// SIMATIC S7-200 project (STEP 7-Micro/WIN), CPU 226 REL 02.01

SYMBOL_TABLE SYM1
ADDR_H           VB102
ADDR_L           VB103
D_H              VB114
D_L              VB115
DATA2_H          VB118
DATA2_L          VB119
DATA1_H          VB120
DATA1_L          VB121
SUM_H            VB122
SUM_L            VB123
SADDR_H          VW202
SADDR_L          VW204
S46H             VW206
S46L             VW208
S51              VW210
S57              VW212
S30_1            VW214
S44              VW216
S30_2            VW218
S30_3            VW220
S30_4            VW222
S30_5            VW224
SD_L             VW226
SD_H             VW228
S30_6            VW230
S31              VW232
SDATA2_H         VW234
SDATA2_L         VW236
SDATA1_H         VW238
SDATA1_L         VW240
END_SYMBOL_TABLE

ORGANIZATION_BLOCK OB_1:OB1
TITLE=【S7-200 PLC与DDM4A数显表的通信控制系统（二）】
// 在生产线上，PLC通过定时器以60个时间周期实现轮询控制。轮询时向分布在不同位置的16个DDM4A数显表发送计数数据，用于显示生产计数和设备状态等关键参数。
// 站点七作为生产线的核心区域，其的DDM4A数显表的计数数据根据实际检测量完成更新。此数据可供其他站点在需要时访问。
// 所有的DDM4A数显表配置为无校验、8位数据、波特率9600bps，使用自由口协议。发送缓冲区长度设为23字节。PLC串口设置和发送缓冲区与之保持一致，以确保通讯正常。
// 在主程序中，首先通过首次扫描设置串口控制字节，启用自由口模式，同时将发送缓冲区长度设为23字节，并初始化轮询控制变量为+1。
// 通过始终为1的位调用轮询子程序。轮询子程序中定时器每60个时间周期触发一次，触发时轮询控制变量左移一位，用于控制轮询。
// 主程序的多个网络分别对应1#站到16#站的发送逻辑。例如，当某站触发信号为真时，设置地址和数据字节，然后调用发送子程序。其他站的逻辑类似，只是地址字节依次递增，最后一站地址使用特定组合。在发送触发网络中，检测各站触发信号的上升沿，任何一位触发时，发送缓冲区开始的23字节数据。
// 在发送子程序中，设置发送缓冲区内容，例如多个命令字节作为固定命令代码。填充字节设为固定值，用于构成数据帧。后续网络将地址字节等转换为整数，存储在变量中，便于计算。校验网络计算SUM校验和，逐步累加所有相关字节的整数值。
// 校验处理网络中，将SUM低字节处理后转换为ASCII码，存储在临时位置，最终设置校验高低字节。
// 轮询子程序的控制网络中，当定时器触发时，轮询控制变量左移一位，实现轮询控制。定时网络中，如果定时器未触发，则启动定时器计时60个周期。
// 数据更新网络中，当站点七触发信号上升沿时，计数变量自增，若达到上限则重置为0，然后将计数变量转换为ASCII码，设置数据字节。
// 站触发信号逐一触发各站发送逻辑。通过触发信号的上升沿检测，确保同一时间只有一个站发送数据。串口配置为无校验、8位数据、波特率9600bps，使用自由口协议，与数显表保持一致。
BEGIN
Network 1
LD     SM0.1
MOVB   16#9, SMB30
MOVB   23, VB100
MOVW   +1, MW1
?000
Network 2
LD     SM0.0
CALL   SBR_1:SBR1
Network 3 // 发送1＃站数据
// 
// 
LD     M1.0
LPS
MOVB   16#31, ADDR_L:VB103
AENO
MOVB   16#30, ADDR_H:VB102
AENO
MOVB   16#30, D_L:VB115
AENO
MOVB   16#30, D_H:VB114
LPP
CALL   SBR_0:SBR0
Network 4 // 发送2＃站数据
// 
// 
LD     M1.1
LPS
MOVB   16#32, ADDR_L:VB103
AENO
MOVB   16#30, ADDR_H:VB102
LPP
CALL   SBR_0:SBR0
Network 5 // 发送3＃站数据
// 
// 
LD     M1.2
LPS
MOVB   16#33, ADDR_L:VB103
AENO
MOVB   16#30, ADDR_H:VB102
LPP
CALL   SBR_0:SBR0
Network 6 // 发送4＃站数据
// 
// 
LD     M1.3
LPS
MOVB   16#34, ADDR_L:VB103
AENO
MOVB   16#30, ADDR_H:VB102
LPP
CALL   SBR_0:SBR0
Network 7 // 发送5＃站数据
// 
// 
LD     M1.4
LPS
MOVB   16#35, ADDR_L:VB103
AENO
MOVB   16#30, ADDR_H:VB102
LPP
CALL   SBR_0:SBR0
Network 8 // 发送6＃站数据
// 
// 
LD     M1.5
LPS
MOVB   16#36, ADDR_L:VB103
AENO
MOVB   16#30, ADDR_H:VB102
LPP
CALL   SBR_0:SBR0
Network 9 // 发送7＃站数据
// 
// 
LD     M1.6
LPS
MOVB   16#37, ADDR_L:VB103
AENO
MOVB   16#30, ADDR_H:VB102
LPP
CALL   SBR_0:SBR0
Network 10 // 发送8＃站数据
// 
// 
LD     M1.7
LPS
MOVB   16#38, ADDR_L:VB103
AENO
MOVB   16#30, ADDR_H:VB102
LPP
CALL   SBR_0:SBR0
Network 11 // 发送9＃站数据
// 
// 
LD     M2.0
LPS
MOVB   16#39, ADDR_L:VB103
AENO
MOVB   16#30, ADDR_H:VB102
LPP
CALL   SBR_0:SBR0
Network 12 // 发送10＃站数据
// 
// 
LD     M2.1
LPS
MOVB   16#41, ADDR_L:VB103
AENO
MOVB   16#30, ADDR_H:VB102
LPP
CALL   SBR_0:SBR0
Network 13 // 发送11＃站数据
// 
// 
LD     M2.2
LPS
MOVB   16#42, ADDR_L:VB103
AENO
MOVB   16#30, ADDR_H:VB102
LPP
CALL   SBR_0:SBR0
Network 14 // 发送12＃站数据
// 
// 
LD     M2.3
LPS
MOVB   16#43, ADDR_L:VB103
AENO
MOVB   16#30, ADDR_H:VB102
LPP
CALL   SBR_0:SBR0
Network 15 // 发送13＃站数据
// 
// 
LD     M2.4
LPS
MOVB   16#44, ADDR_L:VB103
AENO
MOVB   16#30, ADDR_H:VB102
LPP
CALL   SBR_0:SBR0
Network 16 // 发送14＃站数据
// 
// 
LD     M2.5
LPS
MOVB   16#45, ADDR_L:VB103
AENO
MOVB   16#30, ADDR_H:VB102
LPP
CALL   SBR_0:SBR0
Network 17 // 发送15＃站数据
// 
// 
LD     M2.6
LPS
MOVB   16#46, ADDR_L:VB103
AENO
MOVB   16#30, ADDR_H:VB102
LPP
CALL   SBR_0:SBR0
Network 18 // 发送16＃站数据
// 
// 
LD     M2.7
LPS
MOVB   16#30, ADDR_L:VB103
AENO
MOVB   16#31, ADDR_H:VB102
LPP
CALL   SBR_0:SBR0
Network 19 // 发送程序
// 
// 
LD     M1.0
EU
LD     M1.1
EU
OLD
LD     M1.2
EU
OLD
LD     M1.3
EU
OLD
LD     M1.4
EU
OLD
LD     M1.5
EU
OLD
LD     M1.6
EU
OLD
LD     M1.7
EU
OLD
LD     M2.0
EU
OLD
LD     M2.1
EU
OLD
LD     M2.2
EU
OLD
LD     M2.3
EU
OLD
LD     M2.4
EU
OLD
LD     M2.5
EU
OLD
LD     M2.6
EU
OLD
LD     M2.7
EU
OLD
XMT    VB100, 0
END_ORGANIZATION_BLOCK

SUBROUTINE_BLOCK SBR_0:SBR0
TITLE=
BEGIN
Network 1 // 通讯缓冲区 VB102、VB103＝地址；VB114、VB115＝寄存器组；VB118～VB21＝数据；VB122、VB123＝SUM；
LD     SM0.0
MOVB   16#5, VB101
Network 2 // 计算机命令16#46H
//  
LD     SM0.0
MOVB   16#46, VB104
Network 3 // 计算机命令16#46L
//  
LD     SM0.0
MOVB   16#46, VB105
Network 4 // 16#51H
//  
LD     SM0.0
MOVB   16#51, VB106
Network 5 // 16#57
//  
LD     SM0.0
MOVB   16#57, VB107
Network 6 // 16#30
//  
LD     SM0.0
MOVB   16#30, VB108
Network 7 // 16#44
LD     SM0.0
MOVB   16#44, VB109
Network 8 // 16#30
//  
LD     SM0.0
MOVB   16#30, VB110
Network 9 // 16#30
LD     SM0.0
MOVB   16#30, VB111
Network 10 // 16#30
//  
LD     SM0.0
MOVB   16#30, VB112
Network 11 // 16#30
LD     SM0.0
MOVB   16#30, VB113
Network 12 // 16#30
//  
LD     SM0.0
MOVB   16#30, VB116
Network 13 // 16#31
//  
LD     SM0.0
MOVB   16#31, VB117
Network 14 // 将BYTE转换为整形数据，便于计算
LD     SM0.0
BTI    ADDR_L:VB103, SADDR_L:VW204
AENO
BTI    ADDR_H:VB102, SADDR_H:VW202
AENO
BTI    VB104, S46H:VW206
AENO
BTI    VB105, S46L:VW208
Network 15 // 将BYTE转换为整形数据，便于计算
LD     SM0.0
BTI    VB106, S51:VW210
AENO
BTI    VB107, S57:VW212
AENO
BTI    VB108, S30_1:VW214
AENO
BTI    VB109, S44:VW216
Network 16 // 将BYTE转换为整形数据，便于计算
LD     SM0.0
BTI    VB110, S30_2:VW218
AENO
BTI    VB111, S30_3:VW220
AENO
BTI    VB112, S30_4:VW222
AENO
BTI    VB113, S30_5:VW224
Network 17 // 将BYTE转换为整形数据，便于计算
LD     SM0.0
BTI    D_L:VB115, SD_L:VW226
AENO
BTI    D_H:VB114, SD_H:VW228
AENO
BTI    VB116, S30_6:VW230
AENO
BTI    VB117, S31:VW232
Network 18 // 将BYTE转换为整形数据，便于计算
// 
// 
LD     SM0.0
BTI    DATA2_L:VB119, SDATA2_L:VW236
AENO
BTI    DATA2_H:VB118, SDATA2_H:VW234
AENO
BTI    DATA1_L:VB121, SDATA1_L:VW240
AENO
BTI    DATA1_H:VB120, SDATA1_H:VW238
Network 19 // SUM计算
// 
// 
LD     SM0.0
MOVW   SADDR_L:VW204, VW300
AENO
+I     SADDR_H:VW202, VW300
AENO
MOVW   S46H:VW206, VW302
AENO
+I     VW300, VW302
AENO
MOVW   S46L:VW208, VW304
AENO
+I     VW302, VW304
AENO
MOVW   S51:VW210, VW306
AENO
+I     VW304, VW306
AENO
MOVW   S57:VW212, VW308
AENO
+I     VW306, VW308
AENO
MOVW   S30_1:VW214, VW310
AENO
+I     VW308, VW310
AENO
=      M0.0
Network 20
LD     M0.0
MOVW   S44:VW216, VW312
AENO
+I     VW310, VW312
AENO
MOVW   S30_2:VW218, VW314
AENO
+I     VW312, VW314
AENO
MOVW   S30_3:VW220, VW316
AENO
+I     VW314, VW316
AENO
MOVW   S30_4:VW222, VW318
AENO
+I     VW316, VW318
AENO
MOVW   S30_5:VW224, VW320
AENO
+I     VW318, VW320
AENO
MOVW   SD_L:VW226, VW322
AENO
+I     VW320, VW322
AENO
MOVW   SD_H:VW228, VW324
AENO
+I     VW322, VW324
AENO
MOVW   S30_6:VW230, VW326
AENO
+I     VW324, VW326
AENO
=      M0.1
Network 21
LD     M0.1
MOVW   S31:VW232, VW328
AENO
+I     VW326, VW328
AENO
MOVW   SDATA2_L:VW236, VW330
AENO
+I     VW328, VW330
AENO
MOVW   SDATA2_H:VW234, VW332
AENO
+I     VW330, VW332
AENO
MOVW   SDATA1_L:VW240, VW334
AENO
+I     VW332, VW334
AENO
MOVW   SDATA1_H:VW238, VW336
AENO
+I     VW334, VW336
AENO
=      M0.2
Network 22 // ASIC转换为SUM
// 
// 
LD     M0.2
MOVB   VB337, VB340
AENO
ANDB   16#F, VB340
AENO
MOVB   VB337, VB338
AENO
RLB    VB338, 4
AENO
MOVB   VB338, VB341
AENO
ANDB   16#F, VB341
AENO
HTA    VB340, VB270, 4
AENO
MOVB   VB271, SUM_L:VB123
AENO
MOVB   VB273, SUM_H:VB122
END_SUBROUTINE_BLOCK

SUBROUTINE_BLOCK SBR_1:SBR1
TITLE=
BEGIN
Network 1
LD     T32
EU
RLW    MW1, 1
Network 2
LDN    T32
TON    T32, +60
Network 3
LD     M1.7
LPS
EU
INCW   VW250
LRD
AW=    VW250, +10000
MOVW   +0, VW250
LRD
MOVB   VB250, VB256
AENO
ANDB   16#F, VB256
AENO
MOVB   VB250, VB257
AENO
RLB    VB257, 4
AENO
MOVB   VB251, VB258
AENO
ANDB   16#F, VB258
AENO
MOVB   VB251, VB259
AENO
RLB    VB259, 4
AENO
HTA    VB256, VB260, 4
AENO
MOVB   VB263, DATA2_H:VB118
AENO
MOVB   VB261, DATA2_L:VB119
LPP
HTA    VB258, VB265, 4
AENO
MOVB   VB268, DATA1_H:VB120
AENO
MOVB   VB266, DATA1_L:VB121
END_SUBROUTINE_BLOCK
